// Function Block for Delayed Triggers of DIO
FUNCTION_BLOCK FB_Sensor
VAR_INPUT
	Reset			: BOOL;	// Reset Timers/Outputs
	Input			: BOOL;	// Input Status
	OnDelayTime		: TIME;	// Delay to Set On TRUE After Input TRUE
	OffDelayTime	: TIME;	// Delay to Set Off TRUE After Input FALSE
END_VAR

VAR_OUTPUT
	On				: BOOL;	// Status of Delayed Input TRUE
	Off				: BOOL;	// Status of Delayed Input FALSE
END_VAR

VAR
	On_TON			: TON;	// TON Delay for Input TRUE
	Off_TON			: TON;	// TON Delay for Input False
END_VAR


// If Reset Commanded, Reset All
IF Reset THEN
	On_TON(IN := FALSE);
	Off_TON(IN := FALSE);
	On := FALSE;
	Off := FALSE;
	
// Otherwise, Evaluate TONs Based on Input Status
ELSE
	On_TON(
		IN 	:= Input, 
		PT 	:= OnDelayTime,
		Q	=> On);
	
	Off_TON(
		IN 	:= NOT Input, 
		PT 	:= OffDelayTime,
		Q	=> Off);
END_IF;

END_FUNCTION_BLOCK

(* stored: Version 1.1.0.1, ProductVersion 3.1.4024.9
   POU FB_Sensor: Id {dae64110-2125-448a-97a5-670244fb71ad}, SpecialFunc None *)
